(* IEC 61131-3 sources: beckhoffAutomationInterface/ST/Shark/Lib/BehaviorTree/controls, 7 files *)

(* ---- FB_FallbackNode.st ---- *)
FUNCTION_BLOCK FB_FallbackNode IMPLEMENTS I_TreeNode
VAR_INPUT
    sName : STRING(50) := 'Fallback';
END_VAR
VAR
    _list : FB_NodeList;
    _nCurrentChildIndex : INT := 1;
END_VAR

METHOD PUBLIC AddChild : BOOL
VAR_INPUT
    ipNode : I_TreeNode;
END_VAR
    AddChild := _list.AddChild(ipNode);
END_METHOD

METHOD PUBLIC ClearChildren
    _list.ClearChildren();
    _nCurrentChildIndex := 1;
END_METHOD

    {attribute 'estimated-stack-usage' := '500'}
METHOD Tick : ST_NodeResult
VAR
    stChildStatus : ST_NodeResult;
    ipChild       : I_TreeNode;
    sProgressMsg  : STRING(255);
END_VAR

    // If we finished last time, reset to start
    IF _nCurrentChildIndex > _list.GetCount() THEN
        _nCurrentChildIndex := 1;
    END_IF

    WHILE _nCurrentChildIndex <= _list.GetCount() DO

        // Update Progress String for Monitoring
        sProgressMsg := 'Option ';
        sProgressMsg := CONCAT(sProgressMsg, TO_STRING(_nCurrentChildIndex));
        sProgressMsg := CONCAT(sProgressMsg, '/');
        sProgressMsg := CONCAT(sProgressMsg, TO_STRING(_list.GetCount()));

        ipChild := _list.GetChild(_nCurrentChildIndex);

        IF ipChild <> 0 THEN
            stChildStatus := ipChild.Tick();

            sProgressMsg := CONCAT(sProgressMsg, ': ');
            sProgressMsg := CONCAT(sProgressMsg, stChildStatus.sDescription);

            // Blend the running child's own progress with its position so UI
            // moves smoothly, matching FB_SequenceNode / FB_ReactiveSequence.
            Tick.rProgress := F_BlendChildProgress(
                nChildIndex    := _nCurrentChildIndex,
                nTotalChildren := _list.GetCount(),
                rChildProgress := stChildStatus.rProgress
            );
        ELSE
            Tick.eStatus := E_NodeStatus.FAILURE;
            Tick.bHasError := TRUE;
            Tick.stError.eErrorId := E_ErrorId.ERR_BT_NULL_CHILD;
            Tick.stError.sSource := sName;
            Tick.stError.sMessage := CONCAT('Option ', CONCAT(TO_STRING(_nCurrentChildIndex), ' child is null'));
            RETURN;
        END_IF

        IF stChildStatus.eStatus = E_NodeStatus.RUNNING THEN
            Tick.eStatus := E_NodeStatus.RUNNING;
            Tick.sDescription := sProgressMsg;
            RETURN;

        ELSIF stChildStatus.eStatus = E_NodeStatus.SUCCESS THEN
            // Fallback: If one succeeds, the whole node succeeds - clear any errors from previous fallbacks inherently
            Tick.sDescription := 'Done';
            Tick.rProgress := 100.0;
            _nCurrentChildIndex := 1;
            Tick.eStatus := E_NodeStatus.SUCCESS;
            RETURN;

        ELSIF stChildStatus.eStatus = E_NodeStatus.FAILURE THEN
            // Fallback: If one fails, try the next one
            _nCurrentChildIndex := _nCurrentChildIndex + 1;
        END_IF
    END_WHILE

    // If we get here, ALL children failed.
    // stChildStatus already holds the last child's FAILURE result from the loop above —
    // use it directly instead of re-ticking the child, which would issue hardware
    // commands a second time in the same scan cycle.
    IF _list.GetCount() > 0 THEN
        Tick := stChildStatus;  // preserve last child's specific error details
    END_IF
    IF NOT Tick.bHasError THEN
        Tick.bHasError := TRUE;
        Tick.stError.eErrorId := E_ErrorId.ERR_BT_CHILD_FAILED;
        Tick.stError.sSource := sName;
        Tick.stError.sMessage := 'All fallback options failed';
    END_IF

    Tick.eStatus := E_NodeStatus.FAILURE;
    Tick.rProgress := 0.0;
    _nCurrentChildIndex := 1;
END_METHOD

{attribute 'estimated-stack-usage' := '500'}
METHOD Halt
    _list.HaltAll();
    _nCurrentChildIndex := 1;
END_METHOD

{attribute 'estimated-stack-usage' := '500'}
METHOD Reset : BOOL
    _nCurrentChildIndex := 1;
    Reset := _list.ResetAll();
END_METHOD

END_FUNCTION_BLOCK

(* ---- FB_IfThenElseNode.st ---- *)
(* FB_IfThenElseNode — Ternary branch control node

Children:
  Child 1 = Condition
  Child 2 = Then branch
  Child 3 = Else branch

BEHAVIOR:
- Ticks the condition child (1).
- If condition returns SUCCESS → ticks the Then child (2).
- If condition returns FAILURE → ticks the Else child (3).
- If condition returns RUNNING → returns RUNNING.
*)
FUNCTION_BLOCK FB_IfThenElseNode IMPLEMENTS I_TreeNode
VAR_INPUT
    sName : STRING(50) := 'IfThenElse';
END_VAR
VAR
    _list : FB_NodeList;
END_VAR

METHOD PUBLIC AddChild : BOOL
VAR_INPUT
    ipNode : I_TreeNode;
END_VAR
    IF _list.GetCount() >= 3 THEN
        AddChild := FALSE;
        RETURN;
    END_IF
    AddChild := _list.AddChild(ipNode);
END_METHOD

    {attribute 'estimated-stack-usage' := '500'}
METHOD Tick : ST_NodeResult
VAR
    stCondResult : ST_NodeResult;
    stBranchResult : ST_NodeResult;
    ipCondition  : I_TreeNode;
    ipThen       : I_TreeNode;
    ipElse       : I_TreeNode;
END_VAR
    IF _list.GetCount() < 3 THEN
        Tick.eStatus := E_NodeStatus.FAILURE;
        Tick.bHasError := TRUE;
        Tick.stError.eErrorId := E_ErrorId.ERR_BT_NULL_CHILD;
        Tick.stError.sSource := sName;
        Tick.stError.sMessage := 'IfThenElse requires exactly 3 children (condition, then, else)';
        RETURN;
    END_IF

    ipCondition := _list.GetChild(1);
    ipThen      := _list.GetChild(2);
    ipElse      := _list.GetChild(3);

    IF ipCondition = 0 OR ipThen = 0 OR ipElse = 0 THEN
        Tick.eStatus := E_NodeStatus.FAILURE;
        Tick.bHasError := TRUE;
        Tick.stError.eErrorId := E_ErrorId.ERR_BT_NULL_CHILD;
        Tick.stError.sSource := sName;
        Tick.stError.sMessage := 'One or more children are null';
        RETURN;
    END_IF

    // Evaluate condition
    stCondResult := ipCondition.Tick();

    CASE stCondResult.eStatus OF
        E_NodeStatus.SUCCESS:
            stBranchResult := ipThen.Tick();
            Tick := stBranchResult;
            Tick.rProgress := LIMIT(50.0, 50.0 + (stBranchResult.rProgress * 0.5), 100.0);

        E_NodeStatus.FAILURE:
            stBranchResult := ipElse.Tick();
            Tick := stBranchResult;
            Tick.rProgress := LIMIT(50.0, 50.0 + (stBranchResult.rProgress * 0.5), 100.0);

        E_NodeStatus.RUNNING:
            Tick.eStatus := E_NodeStatus.RUNNING;
            Tick.rProgress := LIMIT(0.0, stCondResult.rProgress * 0.5, 50.0);
            Tick.sDescription := 'Evaluating condition';
    ELSE
        Tick.eStatus := E_NodeStatus.FAILURE;
        Tick.bHasError := TRUE;
        Tick.stError.eErrorId := E_ErrorId.ERR_BT_CHILD_FAILED;
        Tick.stError.sSource := sName;
        Tick.stError.sMessage := 'Condition returned unexpected status';
    END_CASE
END_METHOD

{attribute 'estimated-stack-usage' := '500'}
METHOD Halt
    _list.HaltAll();
END_METHOD

{attribute 'estimated-stack-usage' := '500'}
METHOD Reset : BOOL
    Reset := _list.ResetAll();
END_METHOD

END_FUNCTION_BLOCK

(* ---- FB_NodeList.st ---- *)
(* FB_NodeList - Encapsulates child management for composite nodes (Composition over Inheritance). *)
FUNCTION_BLOCK FB_NodeList
VAR
    _aChildren   : ARRAY[1..GVL_BT_Constants.MAX_BT_CHILDREN] OF I_TreeNode;
    _nChildCount : INT := 0;
END_VAR

METHOD PUBLIC AddChild : BOOL
VAR_INPUT
    ipNode : I_TreeNode;
END_VAR
    IF ipNode = 0 THEN
        AddChild := FALSE;
        RETURN;
    END_IF
    IF _nChildCount >= GVL_BT_Constants.MAX_BT_CHILDREN THEN
        AddChild := FALSE;
        RETURN;
    END_IF
    _nChildCount := _nChildCount + 1;
    _aChildren[_nChildCount] := ipNode;
    AddChild := TRUE;
END_METHOD

METHOD PUBLIC ClearChildren
VAR
    i : INT;
END_VAR
    FOR i := 1 TO _nChildCount DO
        _aChildren[i] := 0;
    END_FOR
    _nChildCount := 0;
END_METHOD

METHOD PUBLIC GetChild : I_TreeNode
VAR_INPUT
    nIndex : INT;
END_VAR
    IF nIndex >= 1 AND nIndex <= _nChildCount THEN
        GetChild := _aChildren[nIndex];
    ELSE
        GetChild := 0;
    END_IF
END_METHOD

METHOD PUBLIC GetCount : INT
    GetCount := _nChildCount;
END_METHOD

METHOD PUBLIC HaltAll
VAR
    i : INT;
    ipChild : I_TreeNode;
END_VAR
    FOR i := 1 TO _nChildCount DO
        ipChild := _aChildren[i];
        IF ipChild <> 0 THEN
            ipChild.Halt();
        END_IF
    END_FOR
END_METHOD

METHOD PUBLIC ResetAll : BOOL
VAR
    i : INT;
    ipChild : I_TreeNode;
    bAllReset : BOOL := TRUE;
END_VAR
    FOR i := 1 TO _nChildCount DO
        ipChild := _aChildren[i];
        IF ipChild <> 0 THEN
            IF NOT ipChild.Reset() THEN
                bAllReset := FALSE;
            END_IF
        END_IF
    END_FOR
    ResetAll := bAllReset;
END_METHOD
END_FUNCTION_BLOCK

(* ---- FB_ParallelNode.st ---- *)
(*
FB_ParallelNode
----------------------------------------------------------------------------
PURPOSE:
Executes all children simultaneously every tick.
Succeeds if a required number of children succeed.
Fails if too many children fail such that the required success count is impossible.
----------------------------------------------------------------------------
*)
FUNCTION_BLOCK FB_ParallelNode IMPLEMENTS I_TreeNode
VAR_INPUT
    sName : STRING(50) := 'Parallel Node';
    nSuccessThreshold : INT := -1; // -1 means All
    nFailureThreshold : INT := 1; // Fail on first failure
END_VAR
VAR
    _list : FB_NodeList;
    _aChildStatus : ARRAY[1..GVL_BT_Constants.MAX_BT_CHILDREN] OF E_NodeStatus;
    _nSuccessCount : INT;
    _nFailureCount : INT;
    _bStatusInitialized : BOOL := FALSE;
END_VAR

METHOD PUBLIC AddChild : BOOL
VAR_INPUT
    ipNode : I_TreeNode;
END_VAR
    AddChild := _list.AddChild(ipNode);
END_METHOD

METHOD PUBLIC ClearChildren
    _list.ClearChildren();
    _bStatusInitialized := FALSE;
END_METHOD

    {attribute 'estimated-stack-usage' := '500'}
METHOD Tick : ST_NodeResult
VAR
    i : INT;
    bDone : BOOL;
    ipChild : I_TreeNode;
    stChildStatus : ST_NodeResult;
    rTotalProgress : REAL := 0.0;
    nFirstFailedIdx : INT := 0;
END_VAR

    IF _list.GetCount() <= 0 THEN
        Tick.eStatus := E_NodeStatus.FAILURE;
        Tick.bHasError := TRUE;
        Tick.stError.eErrorId := E_ErrorId.ERR_BT_NULL_CHILD;
        Tick.stError.sSource := sName;
        Tick.stError.sMessage := 'Parallel node has no children configured';
        RETURN;
    END_IF

    IF nFailureThreshold <= 0 THEN
        Tick.eStatus := E_NodeStatus.FAILURE;
        Tick.bHasError := TRUE;
        Tick.stError.eErrorId := E_ErrorId.ERR_GEN_INVALID_PARAM;
        Tick.stError.sSource := sName;
        Tick.stError.sMessage := 'Failure threshold must be greater than zero';
        RETURN;
    END_IF

    IF ((nSuccessThreshold <> -1) AND (nSuccessThreshold <= 0)) OR ((nSuccessThreshold > _list.GetCount()) AND (nSuccessThreshold <> -1)) THEN
        Tick.eStatus := E_NodeStatus.FAILURE;
        Tick.bHasError := TRUE;
        Tick.stError.eErrorId := E_ErrorId.ERR_GEN_INVALID_PARAM;
        Tick.stError.sSource := sName;
        Tick.stError.sMessage := 'Success threshold must be -1 or within child count';
        RETURN;
    END_IF

    IF nFailureThreshold > _list.GetCount() THEN
        Tick.eStatus := E_NodeStatus.FAILURE;
        Tick.bHasError := TRUE;
        Tick.stError.eErrorId := E_ErrorId.ERR_GEN_INVALID_PARAM;
        Tick.stError.sSource := sName;
        Tick.stError.sMessage := 'Failure threshold cannot exceed child count';
        RETURN;
    END_IF

    // Initialize child statuses on first call
    IF NOT _bStatusInitialized THEN
        FOR i := 1 TO GVL_BT_Constants.MAX_BT_CHILDREN DO
            _aChildStatus[i] := E_NodeStatus.IDLE;
        END_FOR
        _bStatusInitialized := TRUE;
    END_IF

    _nSuccessCount := 0;
    _nFailureCount := 0;
    bDone := TRUE;
    Tick.sDescription := 'Running';

    // Tick all children that are not finished
    FOR i := 1 TO _list.GetCount() DO
        ipChild := _list.GetChild(i);
        IF _aChildStatus[i] = E_NodeStatus.IDLE OR _aChildStatus[i] = E_NodeStatus.RUNNING THEN
            IF ipChild <> 0 THEN
                stChildStatus := ipChild.Tick();
                _aChildStatus[i] := stChildStatus.eStatus;

                // Track progress
                rTotalProgress := rTotalProgress + stChildStatus.rProgress;

                // Track first failed child explicitly to bubble up its exact error message
                IF stChildStatus.eStatus = E_NodeStatus.FAILURE AND nFirstFailedIdx = 0 THEN
                     nFirstFailedIdx := i;
                     Tick.stError := stChildStatus.stError; // Copy the inner error
                END_IF
            ELSE
                _aChildStatus[i] := E_NodeStatus.FAILURE;
            END_IF
        ELSE
            // Treat previously finished kids as 100% complete for averaging purposes
            rTotalProgress := rTotalProgress + 100.0;
        END_IF

        IF _aChildStatus[i] = E_NodeStatus.SUCCESS THEN
            _nSuccessCount := _nSuccessCount + 1;
        ELSIF _aChildStatus[i] = E_NodeStatus.FAILURE THEN
            _nFailureCount := _nFailureCount + 1;
        ELSIF _aChildStatus[i] = E_NodeStatus.RUNNING THEN
            bDone := FALSE;
        END_IF
    END_FOR

    // Update Progress
    Tick.rProgress := rTotalProgress / INT_TO_REAL(_list.GetCount());

    // Check thresholds: success when either
    //  - nSuccessThreshold = -1 (meaning 'All') and all children succeeded, or
    //  - nSuccessThreshold > 0 and the success count reached the threshold
    IF
        ( (nSuccessThreshold = -1) AND (_nSuccessCount = _list.GetCount()) )
        OR
        ( (nSuccessThreshold > 0) AND (_nSuccessCount >= nSuccessThreshold) )
        THEN

        // Halt any dynamically remaining children
        _list.HaltAll();

        Tick.eStatus := E_NodeStatus.SUCCESS;
        Tick.sDescription := CONCAT('Succeeded: ', TO_STRING(_nSuccessCount));
        Tick.rProgress := 100.0;

        // Reset initialization flag for next execution
        _bStatusInitialized := FALSE;
        RETURN;
    END_IF

    IF _nFailureCount >= nFailureThreshold THEN

        // Halt any dynamically remaining children
        _list.HaltAll();

        Tick.eStatus := E_NodeStatus.FAILURE;
        Tick.sDescription := CONCAT('Failed: ', TO_STRING(_nFailureCount));
        Tick.bHasError := TRUE;

        // If a child didn't give us a specific error above, generate a wrapper error
        IF Tick.stError.eErrorId = E_ErrorId.NO_ERROR THEN
            Tick.stError.eErrorId := E_ErrorId.ERR_BT_PARALLEL_FAILED;
            Tick.stError.sSource := sName;
            Tick.stError.sMessage := CONCAT(TO_STRING(_nFailureCount), ' parallel children failed');
        END_IF

        _bStatusInitialized := FALSE; // Reset state for future execution
        RETURN;
    END_IF

    IF bDone THEN
        Tick.eStatus := E_NodeStatus.FAILURE;
        Tick.sDescription := 'All children finished without meeting success threshold';
        Tick.bHasError := TRUE;
        Tick.stError.eErrorId := E_ErrorId.ERR_BT_PARALLEL_FAILED;
        Tick.stError.sSource := sName;
        Tick.stError.sMessage := Tick.sDescription;
        _bStatusInitialized := FALSE; // Reset state for future execution
    ELSE
        Tick.eStatus := E_NodeStatus.RUNNING;
    END_IF

END_METHOD

METHOD PRIVATE _ResetState
VAR
    i : INT;
END_VAR
    FOR i := 1 TO GVL_BT_Constants.MAX_BT_CHILDREN DO
        _aChildStatus[i] := E_NodeStatus.IDLE;
    END_FOR
    _nSuccessCount := 0;
    _nFailureCount := 0;
    _bStatusInitialized := FALSE;
END_METHOD

    // Method: Halt - Resets parallel tracking state, halts children
    {attribute 'estimated-stack-usage' := '200'}
{attribute 'estimated-stack-usage' := '500'}
METHOD Halt
    _ResetState();
    _list.HaltAll();
END_METHOD

    {attribute 'estimated-stack-usage' := '200'}
METHOD Reset : BOOL
    _ResetState();
    Reset := _list.ResetAll();
END_METHOD

END_FUNCTION_BLOCK

(* ---- FB_ReactiveSequence.st ---- *)
(*
FB_ReactiveSequence
----------------------------------------------------------------------------
PURPOSE:
Similar to FB_SequenceNode, but re-evaluates all children from the beginning
every tick. Once a child returns RUNNING, it stops execution and returns RUNNING.
If a child returns FAILURE, the sequence fails immediately.
If all children return SUCCESS, the sequence succeeds.

This is highly useful for priority-based behavior where higher priority
conditions/actions must be continuously checked. If a higher priority child
suddenly fails while a lower priority child was running, the sequence reacts
immediately.
----------------------------------------------------------------------------
*)
FUNCTION_BLOCK FB_ReactiveSequence IMPLEMENTS I_TreeNode
VAR_INPUT
    sName : STRING(50) := 'Reactive Sequence';
END_VAR
VAR
    _list : FB_NodeList;
    _nCurrentChildIndex : INT := 1;
END_VAR

METHOD PUBLIC AddChild : BOOL
VAR_INPUT
    ipNode : I_TreeNode;
END_VAR
    AddChild := _list.AddChild(ipNode);
END_METHOD

METHOD PUBLIC ClearChildren
    _list.ClearChildren();
    _nCurrentChildIndex := 1;
END_METHOD

    {attribute 'estimated-stack-usage' := '500'}
METHOD Tick : ST_NodeResult
VAR
    stChildStatus : ST_NodeResult;
    ipChild : I_TreeNode;
    sProgressMsg : STRING(255);
    i : INT;
END_VAR

    // Loop through children starting from index 1 EVERY TICK
    FOR i := 1 TO _list.GetCount() DO

        sProgressMsg := 'Step ';
        sProgressMsg := CONCAT(sProgressMsg, TO_STRING(i));
        sProgressMsg := CONCAT(sProgressMsg, '/');
        sProgressMsg := CONCAT(sProgressMsg, TO_STRING(_list.GetCount()));

        ipChild := _list.GetChild(i);
        IF ipChild <> 0 THEN
            stChildStatus := ipChild.Tick();

            sProgressMsg := CONCAT(sProgressMsg, ': ');
            sProgressMsg := CONCAT(sProgressMsg, stChildStatus.sDescription);

        ELSE
            Tick.eStatus := E_NodeStatus.FAILURE;
            Tick.bHasError := TRUE;
            Tick.stError.eErrorId := E_ErrorId.ERR_BT_NULL_CHILD;
            Tick.stError.sSource := sName;
            Tick.stError.sMessage := CONCAT('Step ', CONCAT(TO_STRING(i), ' child is null'));
            RETURN;
        END_IF

        IF stChildStatus.eStatus = E_NodeStatus.RUNNING THEN
            // If we aborted at a lower index than last cycle, halt the orphaned child
            IF _nCurrentChildIndex > i AND _nCurrentChildIndex <= _list.GetCount() THEN
                ipChild := _list.GetChild(_nCurrentChildIndex);
                IF ipChild <> 0 THEN ipChild.Halt(); END_IF
            END_IF
            _nCurrentChildIndex := i; // Remember where we are currently RUNNING

            Tick.eStatus := E_NodeStatus.RUNNING;
            Tick.sDescription := sProgressMsg;
            Tick.rProgress := F_BlendChildProgress(
                nChildIndex    := i,
                nTotalChildren := _list.GetCount(),
                rChildProgress := stChildStatus.rProgress
            );
            RETURN; // Exit immediately, hold the sequence here for this cycle

        ELSIF stChildStatus.eStatus = E_NodeStatus.FAILURE THEN
            // If we failed at a lower index than the running index from last cycle, halt it
            IF _nCurrentChildIndex > i AND _nCurrentChildIndex <= _list.GetCount() THEN
                ipChild := _list.GetChild(_nCurrentChildIndex);
                IF ipChild <> 0 THEN ipChild.Halt(); END_IF
            END_IF
            _nCurrentChildIndex := 1; // Reset since we failed

            Tick := stChildStatus;
            IF NOT Tick.bHasError THEN
                Tick.bHasError := TRUE;
                Tick.stError.eErrorId := E_ErrorId.ERR_BT_SEQUENCE_FAILED;
                Tick.stError.sSource := sName;
                Tick.stError.sMessage := CONCAT('Failed at step ', TO_STRING(i));
            END_IF
            Tick.sDescription := sProgressMsg;
            RETURN;

        ELSIF stChildStatus.eStatus = E_NodeStatus.SUCCESS THEN
            // Just continue to the next child
            CONTINUE;
        END_IF
    END_FOR

    // If we get here, all children succeeded
    Tick.rProgress := 100.0;
    Tick.sDescription := 'Done';
    _nCurrentChildIndex := 1; // Reset state for future execution
    Tick.eStatus := E_NodeStatus.SUCCESS;
END_METHOD

{attribute 'estimated-stack-usage' := '500'}
METHOD Halt
    _list.HaltAll();
    _nCurrentChildIndex := 1;
END_METHOD

{attribute 'estimated-stack-usage' := '500'}
METHOD Reset : BOOL
    _nCurrentChildIndex := 1;
    Reset := _list.ResetAll();
END_METHOD

END_FUNCTION_BLOCK

(* ---- FB_SequenceNode.st ---- *)
FUNCTION_BLOCK FB_SequenceNode IMPLEMENTS I_TreeNode
VAR_INPUT
    sName : STRING(50) := 'Sequence';
END_VAR
VAR
    _list : FB_NodeList;
    _nCurrentChildIndex : INT := 1;
END_VAR

METHOD PUBLIC AddChild : BOOL
VAR_INPUT
    ipNode : I_TreeNode;
END_VAR
    AddChild := _list.AddChild(ipNode);
END_METHOD

METHOD PUBLIC ClearChildren
    _list.ClearChildren();
    _nCurrentChildIndex := 1;
END_METHOD

    {attribute 'estimated-stack-usage' := '500'}
METHOD Tick : ST_NodeResult
VAR
    stChildStatus : ST_NodeResult;
    ipChild : I_TreeNode;
    sProgressMsg : STRING(255);
END_VAR

    // If we finished last time, reset to start
    IF _nCurrentChildIndex > _list.GetCount() THEN
        _nCurrentChildIndex := 1;
    END_IF

    // Loop through children
    WHILE _nCurrentChildIndex <= _list.GetCount() DO

        // Update Progress String for Monitoring
        sProgressMsg := 'Step ';
        sProgressMsg := CONCAT(sProgressMsg, TO_STRING(_nCurrentChildIndex));
        sProgressMsg := CONCAT(sProgressMsg, '/');
        sProgressMsg := CONCAT(sProgressMsg, TO_STRING(_list.GetCount()));

        ipChild := _list.GetChild(_nCurrentChildIndex);

        IF ipChild <> 0 THEN
            stChildStatus := ipChild.Tick();

            sProgressMsg := CONCAT(sProgressMsg, ': ');
            sProgressMsg := CONCAT(sProgressMsg, stChildStatus.sDescription);

            // Smooth progress
            Tick.rProgress := F_BlendChildProgress(
                nChildIndex    := _nCurrentChildIndex,
                nTotalChildren := _list.GetCount(),
                rChildProgress := stChildStatus.rProgress
            );
        ELSE
            Tick.eStatus := E_NodeStatus.FAILURE;
            Tick.bHasError := TRUE;
            Tick.stError.eErrorId := E_ErrorId.ERR_BT_NULL_CHILD;
            Tick.stError.sSource := sName;
            Tick.stError.sMessage := CONCAT('Step ', CONCAT(TO_STRING(_nCurrentChildIndex), ' child is null'));
            RETURN;
        END_IF

        IF stChildStatus.eStatus = E_NodeStatus.RUNNING THEN
            Tick.eStatus := E_NodeStatus.RUNNING;
            Tick.sDescription := sProgressMsg;
            RETURN;

        ELSIF stChildStatus.eStatus = E_NodeStatus.FAILURE THEN
            // Capture child error and propagate directly
            Tick := stChildStatus;

            IF NOT stChildStatus.bHasError THEN
                // Child failed but didn't set error - create generic error
                Tick.bHasError := TRUE;
                Tick.stError.eErrorId := E_ErrorId.ERR_BT_SEQUENCE_FAILED;
                Tick.stError.sSource := sName;
                Tick.stError.sMessage := CONCAT('Failed at step ', TO_STRING(_nCurrentChildIndex));
            END_IF

            _nCurrentChildIndex := 1;
            Tick.sDescription := sProgressMsg;
            RETURN;

        ELSIF stChildStatus.eStatus = E_NodeStatus.SUCCESS THEN
            _nCurrentChildIndex := _nCurrentChildIndex + 1; // Move to next child
        END_IF
    END_WHILE

    // If we get here, all children succeeded
    Tick.rProgress := 100.0;
    Tick.sDescription := 'Done';
    _nCurrentChildIndex := 1;
    Tick.eStatus := E_NodeStatus.SUCCESS;
END_METHOD

{attribute 'estimated-stack-usage' := '500'}
METHOD Halt
    _list.HaltAll();
    _nCurrentChildIndex := 1;
END_METHOD

{attribute 'estimated-stack-usage' := '500'}
METHOD Reset : BOOL
    _nCurrentChildIndex := 1;
    Reset := _list.ResetAll();
END_METHOD

END_FUNCTION_BLOCK

(* ---- FB_WhileDoElseNode.st ---- *)
(* FB_WhileDoElseNode — While-loop control node

Children:
  Child 1 = Condition
  Child 2 = Do branch (executed while condition succeeds)
  Child 3 = Else branch (executed when condition fails)

BEHAVIOR:
- Ticks the condition child (1).
- If condition returns SUCCESS → ticks the Do child (2).
  - If Do returns RUNNING → returns RUNNING.
  - If Do returns SUCCESS → re-evaluates condition next tick.
  - If Do returns FAILURE → returns FAILURE.
- If condition returns FAILURE → ticks the Else child (3) and returns its result.
- If condition returns RUNNING → returns RUNNING.
*)
FUNCTION_BLOCK FB_WhileDoElseNode IMPLEMENTS I_TreeNode
VAR_INPUT
    sName : STRING(50) := 'WhileDoElse';
END_VAR
VAR
    _list : FB_NodeList;
END_VAR

METHOD PUBLIC AddChild : BOOL
VAR_INPUT
    ipNode : I_TreeNode;
END_VAR
    IF _list.GetCount() >= 3 THEN
        AddChild := FALSE;
        RETURN;
    END_IF
    AddChild := _list.AddChild(ipNode);
END_METHOD

    {attribute 'estimated-stack-usage' := '500'}
METHOD Tick : ST_NodeResult
VAR
    stCondResult : ST_NodeResult;
    ipCondition  : I_TreeNode;
    ipDo         : I_TreeNode;
    ipElse       : I_TreeNode;
END_VAR
    IF _list.GetCount() < 3 THEN
        Tick.eStatus := E_NodeStatus.FAILURE;
        Tick.bHasError := TRUE;
        Tick.stError.eErrorId := E_ErrorId.ERR_BT_NULL_CHILD;
        Tick.stError.sSource := sName;
        Tick.stError.sMessage := 'WhileDoElse requires exactly 3 children (condition, do, else)';
        RETURN;
    END_IF

    ipCondition := _list.GetChild(1);
    ipDo        := _list.GetChild(2);
    ipElse      := _list.GetChild(3);

    IF ipCondition = 0 OR ipDo = 0 OR ipElse = 0 THEN
        Tick.eStatus := E_NodeStatus.FAILURE;
        Tick.bHasError := TRUE;
        Tick.stError.eErrorId := E_ErrorId.ERR_BT_NULL_CHILD;
        Tick.stError.sSource := sName;
        Tick.stError.sMessage := 'One or more children are null';
        RETURN;
    END_IF

    // Evaluate condition
    stCondResult := ipCondition.Tick();

    CASE stCondResult.eStatus OF
        E_NodeStatus.SUCCESS:
            // Condition true → execute Do branch
            Tick := ipDo.Tick();

        E_NodeStatus.FAILURE:
            // Condition false → execute Else branch
            Tick := ipElse.Tick();

        E_NodeStatus.RUNNING:
            Tick.eStatus := E_NodeStatus.RUNNING;
            Tick.sDescription := 'Evaluating condition';
    ELSE
        Tick.eStatus := E_NodeStatus.FAILURE;
        Tick.bHasError := TRUE;
        Tick.stError.eErrorId := E_ErrorId.ERR_BT_CHILD_FAILED;
        Tick.stError.sSource := sName;
        Tick.stError.sMessage := 'Condition returned unexpected status';
    END_CASE
END_METHOD

{attribute 'estimated-stack-usage' := '500'}
METHOD Halt
    _list.HaltAll();
END_METHOD

{attribute 'estimated-stack-usage' := '500'}
METHOD Reset : BOOL
    Reset := _list.ResetAll();
END_METHOD

END_FUNCTION_BLOCK
